(* PLC project Tc2_Utilities.FB_MemRingBuffer Demo, tc3-libraries-kb TwinCAT 3.1 *)
(* stored: creationDateTime 2026-05-10T20:00:00, modificationDateTime 2026-05-10T20:00:00 *)

PROGRAM P_Demo_FB_MemRingBuffer
  VAR
    fbFB_MemRingBuffer : FB_MemRingBuffer;  (* Tc2_Utilities.FB_MemRingBuffer 实例 *)
    arg_pWrite : POINTER TO BYTE;  (* VAR_INPUT pWrite *)
    arg_cbWrite : UDINT;  (* VAR_INPUT cbWrite *)
    arg_pRead : POINTER TO BYTE;  (* VAR_INPUT pRead *)
    arg_cbRead : UDINT;  (* VAR_INPUT cbRead *)
    arg_pBuffer : POINTER TO BYTE;  (* VAR_INPUT pBuffer *)
    arg_cbBuffer : UDINT;  (* VAR_INPUT cbBuffer *)
    out_bOk : BOOL;  (* VAR_OUTPUT bOk *)
    out_nCount : UDINT;  (* VAR_OUTPUT nCount *)
    out_cbSize : UDINT;  (* VAR_OUTPUT cbSize *)
    out_cbReturn : UDINT;  (* VAR_OUTPUT cbReturn *)
  END_VAR

            // ============================================================
// Tc2_Utilities.FB_MemRingBuffer 演示程序（FB 实例）
// ============================================================
// 验证步骤：
//   1. 引用 Tc2_Utilities（及依赖类型所在库 Tc2_System 等）
//   2. 编译 + 登录
//   3. 按 doc.md 给 arg_* 赋值
//   4. 在线监视 out_* / io_* 输出
// ============================================================

fbFB_MemRingBuffer(
    pWrite := arg_pWrite,
    cbWrite := arg_cbWrite,
    pRead := arg_pRead,
    cbRead := arg_cbRead,
    pBuffer := arg_pBuffer,
    cbBuffer := arg_cbBuffer,
    bOk => out_bOk,
    nCount => out_nCount,
    cbSize => out_cbSize,
    cbReturn => out_cbReturn
);

          
END_PROGRAM
